{attribute 'GeneratedUsingTerminal: KL3051'}
{attribute addProperty BoxType "KL3051"}
{attribute addProperty Id "Channel_1AT %Q*Channel_6576A6810"}
{attribute addProperty CRC "1632160004"}
{attribute addProperty Size "0"}
TYPE KL3051_6148C904 :
STRUCT
	{attribute addProperty Name "Channel_1"}
	Channel_1 : Channel_6576A681;
END_STRUCT
END_TYPE

(* stored: Version 1.2.0.0, ProductVersion 3.1.4024.9
   DUT KL3051_6148C904: Id {5d78ea17-1e2d-4f53-ae48-34afb47a6fc9} *)
